{attribute 'qualified_only'}
{attribute 'strict'}
{attribute 'to_string'}
TYPE E_MoverTask :
(
IDLE :=0,
JOIN,
MOVE_TRACK,
MOVE_C_ROTATE,
RESET_ROTATE,
RESET_ERROR
);
END_TYPE

(* stored: Version 1.1.0.1
   DUT E_MoverTask: Id {950b3f6c-c276-4d7f-ae8c-291149e11350} *)
